TYPE DUT_SequenceByName :
STRUCT
	return_value	: DINT;
	SequenceName	: STRING(50);
END_STRUCT
END_TYPE

(* stored: Version 1.1.0.1, ProductVersion 3.1.4024.15
   DUT DUT_SequenceByName: Id {3e278516-021d-4091-8298-e98f44c00498} *)
